FUNCTION ifExprFunc1 : LREAL
VAR_INPUT
	state: STATE;
END_VAR

IF ((state.dvar_M_example_controller) = (elit_init2)) THEN
    ifExprFunc1 := 0.0;
ELSIF ((state.dvar_M_example_controller) = (elit_wait_start)) THEN
    ifExprFunc1 := 0.0;
ELSIF ((state.dvar_M_example_controller) = (elit_reset_button)) THEN
    ifExprFunc1 := 0.0;
ELSIF ((state.dvar_M_example_controller) = (elit_pauze_left)) THEN
    ifExprFunc1 := 0.0;
ELSIF ((state.dvar_M_example_controller) = (elit_wait_vacuum)) THEN
    ifExprFunc1 := 0.0;
ELSIF ((state.dvar_M_example_controller) = (elit_reset_down)) THEN
    ifExprFunc1 := 0.0;
ELSIF ((state.dvar_M_example_controller) = (elit_reset_place)) THEN
    ifExprFunc1 := 0.0;
ELSIF ((state.dvar_M_example_controller) = (elit_droppoint)) THEN
    ifExprFunc1 := 0.0;
ELSIF ((state.dvar_M_example_controller) = (elit_movetopickup)) THEN
    ifExprFunc1 := 0.0;
ELSIF ((state.dvar_M_example_controller) = (elit_down)) THEN
    ifExprFunc1 := 0.0;
ELSIF ((state.dvar_M_example_controller) = (elit_gopickup)) THEN
    ifExprFunc1 := 0.0;
ELSIF ((state.dvar_M_example_controller) = (elit_goback)) THEN
    ifExprFunc1 := 1.0;
ELSIF ((state.dvar_M_example_controller) = (elit_finished)) THEN
    ifExprFunc1 := 0.0;
ELSE
    ifExprFunc1 := 1.0;
END_IF;

END_FUNCTION

(* stored: Version 1.1.0.1, ProductVersion 3.1.4022.18
   POU ifExprFunc1: Id {34d0acb7-8de3-41a4-a4d8-5299e538b73f}, SpecialFunc None *)
